(* CoDeSys 2.3 export: ATTR3_TU.EXP *)

(* Data type in Diag/Parameter *)
TYPE attr3_tu :
STRUCT
	StepWidth_u16			: UINT;
(*
	FunctionNumber_u16	: UINT;
	FrequencyRange_u16	: UINT;
	data_au8 				: ARRAY [1..2] OF USINT;
*)
END_STRUCT
END_TYPE
